% RSLogix 500 project BITWISENAND_BAK081.RSS, saved by version 8.30.00.16 %
PROJECT "UNTITLED"    % processor: MicroLogix 1000 %

PROGRAM FILES
  LAD 2 "MAIN_PROG"  7 rungs
  LAD 3 "USER_FAULT"  1 rungs
  LAD 4 "HSC_INT"  1 rungs
  LAD 5 "STI_INT"  1 rungs
  LAD 6, 7, 8, 9, 10, 11, 12, 13, 14, 15, 16: only END

DATA FILES
  O0 OUTPUT  1 elements
  I1 INPUT  2 elements
  S2 STATUS  33 elements
  B3 BINARY  32 elements
  T4 TIMER  40 elements
  C5 COUNTER  32 elements
  R6 CONTROL  16 elements
  N7 INTEGER  105 elements

LADDER 2 "MAIN_PROG"
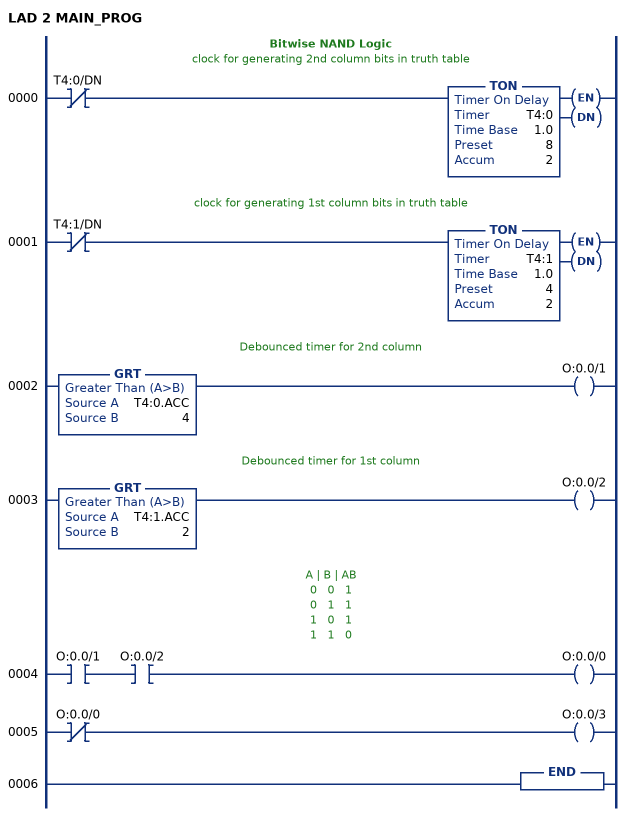
% Rung: 0 %
% TITLE: Bitwise NAND Logic %
% clock for generating 2nd column bits in truth table %
SOR XIO T4:0/DN TON T4:0 1.0 8 2 EOR
% Rung: 1 %
% clock for generating 1st column bits in truth table %
SOR XIO T4:1/DN TON T4:1 1.0 4 2 EOR
% Rung: 2 %
% Debounced timer for 2nd column %
SOR GRT T4:0.ACC 4 OTE O:0.0/1 EOR
% Rung: 3 %
% Debounced timer for 1st column %
SOR GRT T4:1.ACC 2 OTE O:0.0/2 EOR
% Rung: 4 %
% A | B | AB
% 0   0   1
% 0   1   1
% 1   0   1
% 1   1   0 %
SOR XIC O:0.0/1 XIC O:0.0/2 OTE O:0.0/0 EOR
% Rung: 5 %
SOR XIO O:0.0/0 OTE O:0.0/3 EOR
% Rung: 6 %
SOR END EOR

DATA TABLE (non-zero values as saved)
DATA B3
% B3:0 % 0X000F 0X0000 0X0000 0X0000 0X0000 0X0000 0X0000 0X0000 0X0000 0X0000
DATA T4
% .PRE .ACC %
% T4:0 % 8 2
% T4:1 % 4 2
